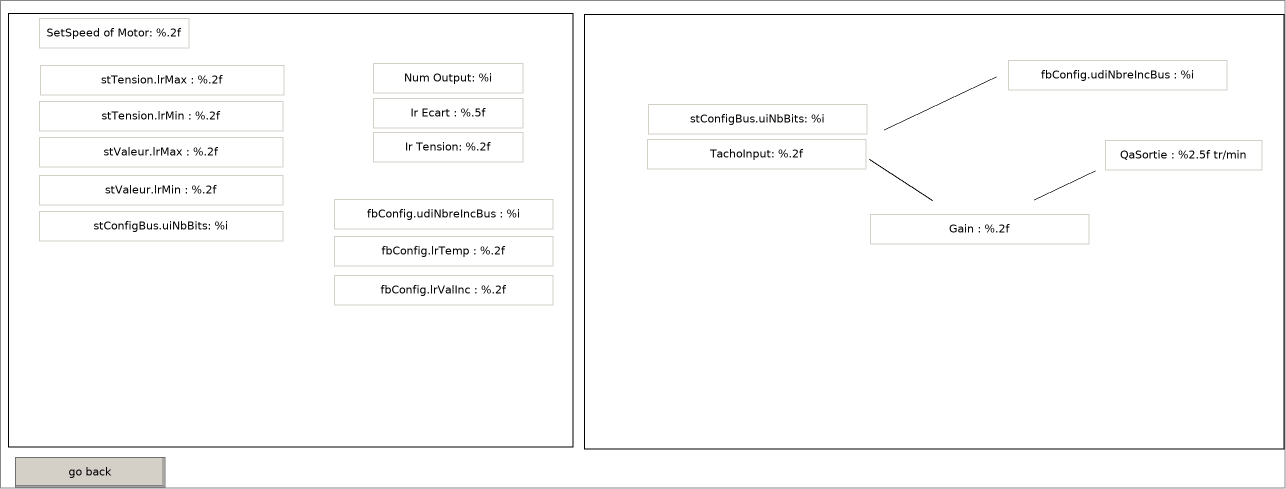
VISUALIZATION VisuMotor  // 1286x489
    Group (160,59 240x84)
        Label (0,0 237x66), "You are not allowed to see this page"
        Label (3,18 237x66), "Please login as another user"
    Rectangle (8,13 565x434)
    Rectangle (584,14 700x435)
    Button (15,457 150x30), "go back", text list: ''
        OnMouseClick: change screen: Visualization
    Line (869,159) (932,200)
    Line (1095,171) (1034,200)
    Line (996,77) (884,130)
    Textfield (373,98 150x30), "Ir Ecart : %.5f", text variable: fbMotor.fbConvertNumToMotorOut.lrEcart
    Textfield (373,132 150x30), "Ir Tension: %.2f", text variable: fbMotor.fbConvertNumToMotorOut.lrTension
    Textfield (40,65 244x30), "stTension.lrMax : %.2f", text variable: fbMotor.fbConvertNumToMotorOut.fbConfig.stTension.lrMax
        OnMouseClick: write the text variable via Default
    Textfield (39,18 150x30), "SetSpeed of Motor: %.2f", text variable: fbMotor.fbConvertNumToMotorOut.lrConsigne
    Textfield (39,101 244x30), "stTension.lrMin : %.2f", text variable: fbMotor.fbConvertNumToMotorOut.fbConfig.stTension.lrMin
        OnMouseClick: write the text variable via Default
    Textfield (39,137 244x30), "stValeur.lrMax : %.2f", text variable: fbMotor.fbConvertNumToMotorOut.fbConfig.stValeur.lrMax
        OnMouseClick: write the text variable via Default
    Textfield (39,175 244x30), "stValeur.lrMin : %.2f", text variable: fbMotor.fbConvertNumToMotorOut.fbConfig.stValeur.lrMin
        OnMouseClick: write the text variable via Default
    Textfield (39,211 244x30), "stConfigBus.uiNbBits: %i", text variable: fbMotor.fbConvertNumToMotorOut.fbConfig.uiNbreBitBus
        OnMouseClick: write the text variable via Default
    Textfield (334,199 219x30), "fbConfig.udiNbreIncBus : %i", text variable: fbMotor.fbConvertNumToMotorOut.fbConfig.udiNbreIncBus
        OnMouseClick: write the text variable via Default
    Textfield (334,236 219x30), "fbConfig.lrTemp : %.2f", text variable: fbMotor.fbConvertNumToMotorOut.fbConfig.lrTemp
        OnMouseClick: write the text variable via Default
    Textfield (334,275 219x30), "fbConfig.lrValInc : %.2f", text variable: fbMotor.fbConvertNumToMotorOut.fbConfig.lrValInc
        OnMouseClick: write the text variable via Default
    Textfield (648,104 219x30), "stConfigBus.uiNbBits: %i", text variable: fbMotor.fbConvertTachoToNumSpeed.fbConfig.uiNbreBitBus
        OnMouseClick: write the text variable via Default
    Textfield (647,139 219x30), "TachoInput: %.2f", text variable: fbMotor.fbConvertTachoToNumSpeed.IaEntree
        OnMouseClick: write the text variable via Default
    Textfield (1105,140 157x30), "QaSortie : %2.5f tr/min", text variable: fbMotor.fbConvertTachoToNumSpeed.lrValeur
        OnMouseClick: write the text variable via Default
    Textfield (870,214 219x30), "Gain : %.2f", text variable: fbMotor.fbConvertTachoToNumSpeed.fbConfig.stValeur.lrMax
        OnMouseClick: write the text variable via Default
    Textfield (1008,60 219x30), "fbConfig.udiNbreIncBus : %i", text variable: fbMotor.fbConvertTachoToNumSpeed.fbConfig.uiNbreBitBus
        OnMouseClick: write the text variable via Default
    Textfield (373,63 150x30), "Num Output: %i", text variable: fbMotor.fbConvertNumToMotorOut.QaSortie
        OnMouseClick: write the text variable via Default
END_VISUALIZATION

(* stored: Version 1.1.0.1, ProductVersion 3.1.4020.6
   Visu VisuMotor: Id {263718a9-e13e-4e85-8a48-6b2945f8f0a0} *)
